{attribute wpf [Container(Layout.Wrap)]}
TYPE WrapLayout:
STRUCT
	_various_types: VariousTypes;
END_STRUCT
END_TYPE

(* stored: Version 1.1.0.1, ProductVersion 3.1.4024.9
   DUT WrapLayout: Id {9d7ec322-52e6-4d4e-997b-911c98c9627a} *)
